INTERFACE I_GantryPart

PROPERTY PartPicked : BOOL
GET
END_GET
END_PROPERTY

PROPERTY PartReady : BOOL
GET
END_GET
END_PROPERTY

END_INTERFACE

(* stored: Version 1.1.0.1, ProductVersion 3.1.4024.4
   Itf I_GantryPart: Id {c3f1e846-cf22-4441-911d-82affc0b3f71}
   Property PartPicked: Id {ff0c925f-c073-4dbe-a44b-3bdecc4b0a18}
   Get Get: Id {d8dd96f9-71e8-4bae-a830-60376042fdeb}
   Property PartReady: Id {225ba40e-ba68-419f-b5e2-445abf6deedc}
   Get Get: Id {2ae7c79e-0ac1-4342-9138-7900329562cc} *)
